Staubli VAL3: debug.pgx

public program debug(num& x_nExecStatus)
begin

  // Debug

  gotoxy(scMonitor, 18,12)
  switch x_nExecStatus
    case 0
      put(scMonitor, "[+]")
      x_nExecStatus = 1
    break
    case 1
      put(scMonitor, "[-]")
      x_nExecStatus = 0
    break
    default
    break
  endSwitch

end
